// TIA Portal V20 export
DATA_BLOCK "Config"   // DB93
// stored: MemoryReserve 100, Namespace Unit1.Em9
   VAR
      em : "LAF_typeEmConfiguration";   // Configuration of EM Parameters
      cmVisionJRDetect : "LBC_typeDigitalSignalConfiguration";
      cmVisionStageLiftUpDown : "LBC_typeTwoWayActuatorConfiguration";
      cmVisionLightUpDown : "LBC_typeTwoWayActuatorConfiguration";
      cmVisionControl : "LER_typeVisionConfiguration";
   END_VAR
BEGIN
   em.referenceDesignator.parent := WSTRING#'U1';
   em.referenceDesignator.relative := WSTRING#'EM0';
   cmVisionStageLiftUpDown.referenceDesignator := WSTRING#'FINAL VISION STAGE LIFT';
   cmVisionStageLiftUpDown.monitoringDiscrepancy := T#5s;
   cmVisionLightUpDown.referenceDesignator := WSTRING#'FINAL VISION LIGHT';
   cmVisionLightUpDown.monitoringDiscrepancy := T#5s;
   cmVisionControl.hwID.cmdResultStatusID := 1015;
   cmVisionControl.hwID.trgReadyStatusID := 1016;
   cmVisionControl.hwID.trgAckStatusID := 1017;
   cmVisionControl.hwID.miscellaneousStatusID := 1018;
   cmVisionControl.hwID.assignableStatusID := 1019;
   cmVisionControl.hwID.resultData248ByteID_1 := 1020;
   cmVisionControl.hwID.resultData248ByteID_2 := 1020;
   cmVisionControl.hwID.resultData248ByteID_3 := 1020;
   cmVisionControl.hwID.resultData248ByteID_4 := 1020;
   cmVisionControl.hwID.resultData248ByteID_5 := 1020;
   cmVisionControl.hwID.cmdResultControlID := 1021;
   cmVisionControl.hwID.trgControlID := 1022;
   cmVisionControl.hwID.miscellaneousControlID := 1023;
   cmVisionControl.hwID.reservedControlID := 1024;
   cmVisionControl.hwID.assignableControlID := 1025;
   cmVisionControl.hwID.parameterData248ByteID_1 := 1026;
   cmVisionControl.hwID.parameterData248ByteID_2 := 258;
   cmVisionControl.hwID.parameterData248ByteID_3 := 260;
   cmVisionControl.hwID.parameterData248ByteID_4 := 261;
   cmVisionControl.hwID.parameterData248ByteID_5 := 262;
   cmVisionControl.trigger1Use := TRUE;
   cmVisionControl.triggertime := T#500ms;
   cmVisionControl.cycleTime := T#5s;
END_DATA_BLOCK
